TYPE enBOT_API :
(
	none := 0, getMe := 1, sendMsg := 2, getUpdates := 3
);
END_TYPE

(* stored: Version 1.1.0.1, ProductVersion 3.1.4024.12
   EnumerationTextList enBOT_API: Id {9e00ccc2-7ec7-492a-9077-9a32d3570811} *)
